# EPICS substitutions: mpexApp/Db/vac_pmi.substitutions
file "valve.db" {
    pattern { SYS, SDEV }
    { "VAC_PMI", "TTRAIN" }
}

file "gauge.db" {
    pattern { SYS }
    { "VAC_PMI" }
}
